FUNCTION F_IsFunctionErrorPending : BOOL
(**************************************************************************************
 * 	Application		:	BoxControl Framework
 *	Revision		:	$Revision: 404529 $
 *	Revision date	:	$Date: 2018-04-23 08:21:38 +0200 (Mo., 23 Apr 2018) $
 *	Last changed by	:	$Author: b7bolm $
 *	URL				:	$URL: http://almscdc.swisslog.com/repo/SWPD/Development/BoxControlFramework/20_Release/trunk/01_Software/BCF/BCF/JumpStart/20_Product/10_App/12_E_Functions/10_Lib/10_Conv/10_Functions/F_IsFunctionErrorPending.TcPOU $
 *
 *	Purpose			:	Check if an error is pending on function and its containing zones
 *
 * ------------------------------------------------------------------------------------
 *	Copyright Swisslog [IP AG], Switzerland. All rights reserved.
 * 
 * ------------------------------------------------------------------------------------
 *	
 * 	Revision History: 
 *
 * 	VERSION			DATE			INITIALS			DESCRIPTION
 *	0.1				01.01.2001		swl					Example
 *
 **************************************************************************************)
VAR_INPUT
	eFunctionNumber		: E_FunctionNumber; // Function number
END_VAR

// Initialize
F_IsFunctionErrorPending := FALSE;

// Check if element number is valid
IF eFunctionNumber > E_FunctionNumber.F_BEGIN_FUNCTION AND
   eFunctionNumber < E_FunctionNumber.F_END_FUNCTION THEN

	// Check reference is valid
	IF __ISVALIDREF(FunctionRegistry[eFunctionNumber].rFunctionData) THEN
   		// Return error state
   		F_IsFunctionErrorPending := FunctionRegistry[eFunctionNumber].rFunctionData.ErrorData.Error.ErrorType = E_ErrorType.ERROR OR
									FunctionRegistry[eFunctionNumber].rFunctionData.ErrorData.ZoneErrorPending;
	END_IF
END_IF

END_FUNCTION

(* stored: Version 1.1.0.1, ProductVersion 3.1.4022.12
   POU F_IsFunctionErrorPending: Id {c6f0f9a8-1d42-46d7-8347-f1f15b1d6509}, SpecialFunc None *)
